TYPE ST_PneumaticAxisStatus :
STRUCT
    bExtendMoving: BOOL; //Extraction movement status
    bRetractMoving: BOOL; //Retraction movement status
    bExtractedStatus: BOOL; //Cylinder extracted status
    bRetractedStatus: BOOL; //Cylinder retracted status
    sStatus: STRING; //Pneumatic cylinder current status
    bErrorStatus: BOOL; //Pneumatic axis is in Error state
END_STRUCT
END_TYPE

(* stored: Version 1.1.0.1, ProductVersion 3.1.4024.5
   DUT ST_PneumaticAxisStatus: Id {7869817a-a6d6-4657-92fd-c307a4cba7d6} *)
